(* Logix 5000 project; controller PLC vendor 1 type 14 code 155 rev 30.14; software revision 30.01; part 5 of 5 *)
(* tags used below, declared in another part *)
   Denester : Denester_R2b;
   Denester_index_counter : COUNTER;
   HMI_Enable_Denester : BOOL;
   IO : IO_R2a;
   OS : INT[10];
   System : System_R2e;
   Test_Bits : BOOL[32];
   Ulma_Running_Bypass : BOOL;
(* MainProgram, continued *)

ROUTINE File_300_Denester   (* ladder *)
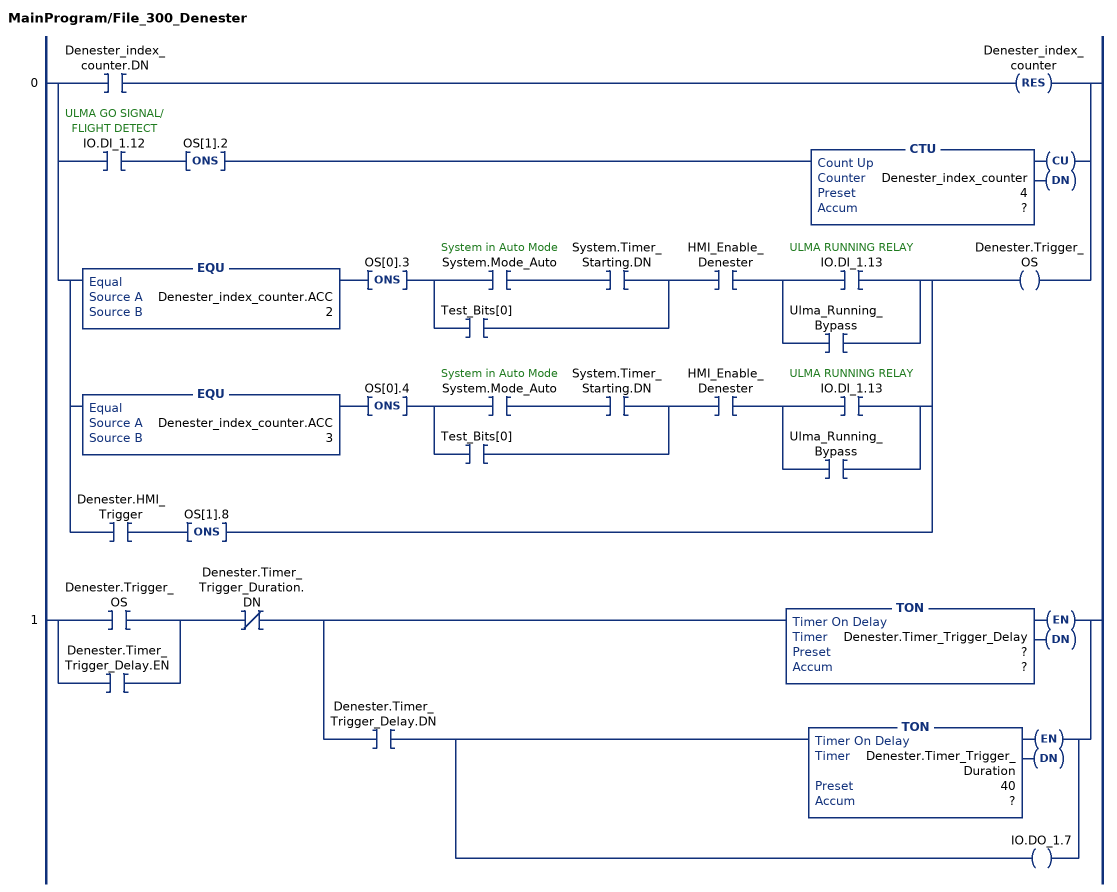
   0: [XIC(Denester_index_counter.DN) RES(Denester_index_counter) ,XIC(IO.DI_1.12) ONS(OS[1].2) CTU(Denester_index_counter,?,?) ,[EQU(Denester_index_counter.ACC,2) ONS(OS[0].3) [XIC(System.Mode_Auto) XIC(System.Timer_Starting.DN) ,XIC(Test_Bits[0]) ] XIC(HMI_Enable_Denester) [XIC(IO.DI_1.13) ,XIC(Ulma_Running_Bypass) ] ,EQU(Denester_index_counter.ACC,3) ONS(OS[0].4) [XIC(System.Mode_Auto) XIC(System.Timer_Starting.DN) ,XIC(Test_Bits[0]) ] XIC(HMI_Enable_Denester) [XIC(IO.DI_1.13) ,XIC(Ulma_Running_Bypass) ] ,XIC(Denester.HMI_Trigger) ONS(OS[1].8) ] OTE(Denester.Trigger_OS) ];
   1: [XIC(Denester.Trigger_OS) ,XIC(Denester.Timer_Trigger_Delay.EN) ]XIO(Denester.Timer_Trigger_Duration.DN)[TON(Denester.Timer_Trigger_Delay,?,?) ,XIC(Denester.Timer_Trigger_Delay.DN) [TON(Denester.Timer_Trigger_Duration,?,?) ,OTE(IO.DO_1.7) ] ];
END_ROUTINE
END_PROGRAM
